(* IEC 61131-3 sources: CodesysTest/export/UN00 - Sharp Bagger/EM01 - Bagger Head/CM05 - Printer/FB_BasicPrinter.pou, 2 files *)

(* ---- FB_BasicPrinter.pou.st ---- *)
(*#-#-#-#-#-#-#-#-#-#---Declaration---#-#-#-#-#-#-#-#-#-#-#-#-#*)

FUNCTION_BLOCK FB_BasicPrinter EXTENDS FB_BaseComponent IMPLEMENTS IPrinter, ISimulateable
VAR_INPUT
	simulateIO : BOOL;
	printSpeed : UDINT;
	printLength : REAL;
END_VAR
VAR_OUTPUT
END_VAR
VAR
	_hasLabel : BOOL;
	_printDone : BOOL;
	_beginPrinting : BOOL;
	_stopPrinting : BOOL;
	_printing : BOOL;
	_simulate : BOOL;
	state : eZebraPrinterStates;;
END_VAR
(*#-#-#-#-#-#-#-#-#-#---Implementation---#-#-#-#-#-#-#-#-#-#-#-#-#*)

SUPER^();

(* ---- StopPrinting.m.st ---- *)
(*#-#-#-#-#-#-#-#-#-#---Declaration---#-#-#-#-#-#-#-#-#-#-#-#-#*)

METHOD StopPrinting
VAR_INPUT
END_VAR
(*#-#-#-#-#-#-#-#-#-#---Implementation---#-#-#-#-#-#-#-#-#-#-#-#-#*)

_stopPrinting := TRUE;
